FUNCTION_BLOCK E_IMPULSE (* Composite FB wrapping other FBs *)
  (* Standard: 61499-2 *)
  (* Version 1.0, 2022-11-09, franz *)
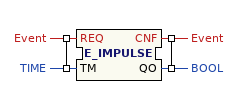
  EVENT_INPUT
    REQ WITH TM; (* Normal Execution Request *)
  END_EVENT
  EVENT_OUTPUT
    CNF WITH QO; (* Execution Confirmation *)
  END_EVENT
  VAR_INPUT
    TM : TIME;
  END_VAR
  VAR_OUTPUT
    QO : BOOL; (* Output event qualifier *)
  END_VAR
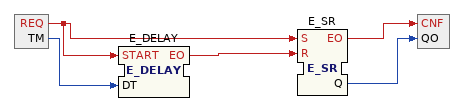
  FBS
    E_DELAY : E_DELAY;
    E_SR : E_SR;
  END_FBS
  EVENT_CONNECTIONS
    REQ TO E_DELAY.START;
    REQ TO E_SR.S;
    E_DELAY.EO TO E_SR.R;
    E_SR.EO TO CNF;
  END_CONNECTIONS
  DATA_CONNECTIONS
    TM TO E_DELAY.DT;
    E_SR.Q TO QO;
  END_CONNECTIONS
END_FUNCTION_BLOCK
